(* PLC project Untitled1, Beckhoff Automation GmbH TF6420 Database Server Query Analyser 1.0.0.0 *)
(* stored: creationDateTime 2016-04-21T11:41:57, modificationDateTime 2016-04-21T11:41:57 *)

TYPE DB_r134a : STRUCT
  id : DINT;
  timestamp : DT;
  Temperatur : STRING(45);
  Enthalpie : STRING(45);
  Druck : STRING(45);
END_STRUCT;
END_TYPE
